INTERFACE I_Link EXTENDS I_Disposable

PROPERTY PUBLIC Id : T_MAXSTRING
GET
END_GET
END_PROPERTY

END_INTERFACE

(* stored: Version 1.1.0.1, ProductVersion 3.1.4024.12
   Itf I_Link: Id {a05f45a8-52a5-02b5-01cd-9cccba704f4c}
   Property Id: Id {d8a1d51f-1ef7-0750-288e-3d562c7c9a77}
   Get Get: Id {e6bbada7-049b-08ca-27aa-960c04438e92} *)
